FUNCTION_BLOCK ABSTRACT AbstractReceiver IMPLEMENTS I_Callable, I_Receiver
VAR
	_tag: Tag;
END_VAR

(*
This method provides a standardized way for other objects to interact with the object that owns it.
*)
METHOD Call
VAR_INPUT
	iArg	: I_Arg;
END_VAR
END_METHOD

METHOD INTERNAL Receive
VAR_INPUT
	iArg			: I_Arg;
END_VAR
Call(iArg);
END_METHOD

(*
Provides access to the tag associated with the signal.
*)
PROPERTY FINAL Tag : I_Tag
GET
Tag := _tag;
END_GET
END_PROPERTY

END_FUNCTION_BLOCK

(* stored: Version 1.1.0.1
   POU AbstractReceiver: Id {c46f739c-8b3f-4cdd-8554-e44831648382}, SpecialFunc None
   Method Call: Id {7bd0ae8b-60bb-4ea9-8cdc-b0909f6a307e}
   Method Receive: Id {952bece5-ce03-46c2-9fe8-6d4fb98ee01d}
   Property Tag: Id {bf34ea37-dbe0-4dda-85a8-706b9379267c}
   Get Get: Id {904ebb0a-3e09-4e22-b46c-582b44ddc0fb} *)
